(* general cam lock ctrl *)
FUNCTION_BLOCK FB_MC2_CamCtrl
VAR_INPUT
	bLockCam			: BOOL;			(* set TRUE to lock Slave axis to Master axis using cam table *)
	eStartMode			: MC_StartMode;	(* start mode for cam *)
	eCamTableID			: MC_CAM_ID;	(* NC cam table ID *)
	sCamTableRef		: MC_CAM_REF;	(* cam table reference structure *)
	fMasterOffset		: LREAL;		(* master offset on cam lock *)
	fSlaveOffset		: LREAL;		(* slave offset on cam lock *)
	fMasterScaling		: LREAL;		(* master scaling *)
	fSlaveScaling		: LREAL;		(* slave scaling *)
	sCamInOptions		: ST_CamInOptions;	(* cam coupling options *)
END_VAR
VAR_IN_OUT
	sMasterAxis			: AXIS_REF;		(* master axis *)
	sSlaveAxis			: AXIS_REF;		(* slave axis *)
END_VAR
VAR_OUTPUT
	bCamLocked			: BOOL;			(* TRUE = cam locked *)
	bCamError			: BOOL;			(* TRUE = cam lock error *)
	nCamErrorID			: UDINT;		(* cam lock error code *)
	bCamTableReadOK		: BOOL;			(* TRUE = cam table loaded from NC *)
	bCamActive			: BOOL;			(* TRUE = cam plate active but not yet in use *)
	bCamInSync			: BOOL;			(* TRUE = cam plate active and in use *)
	bCamUnlockPulse		: BOOL;			(* TRUE = cam has been unlocked, one-shout pulse output *)
	nCamPoints			: UDINT;		(* no of cam points in NC cam table *)
	sCamInfo			: MC_CamInfoData;	(* cam info *)
END_VAR
VAR
	fbPhaseDelay		: TON;
	fbReadCamTable		: MC_ReadMotionFunction;
	fbEnableCamLock		: RS;
	bEnableCamLock		: BOOL;
	fbLockCam			: MC_CamIn;
	fbUnlockCam			: MC_CamOut;
	bCamReady			: BOOL;
	fbCamInfo			: MC_CamInfo;
	bCamInfoDone		: BOOL;
	fbUnlockEvent		: F_TRIG;
	fbUnlockPulse		: TP;
END_VAR
(*
-------------------------------------------------------------------------------------------------
Date		Version	Author	Comments
-------------------------------------------------------------------------------------------------
30/01/2015	3.00.00	PB		Initial release

-------------------------------------------------------------------------------------------------
*)
VAR // added by the converter: edge detectors and wires of the graphical bodies
    _w1 : BOOL;
END_VAR

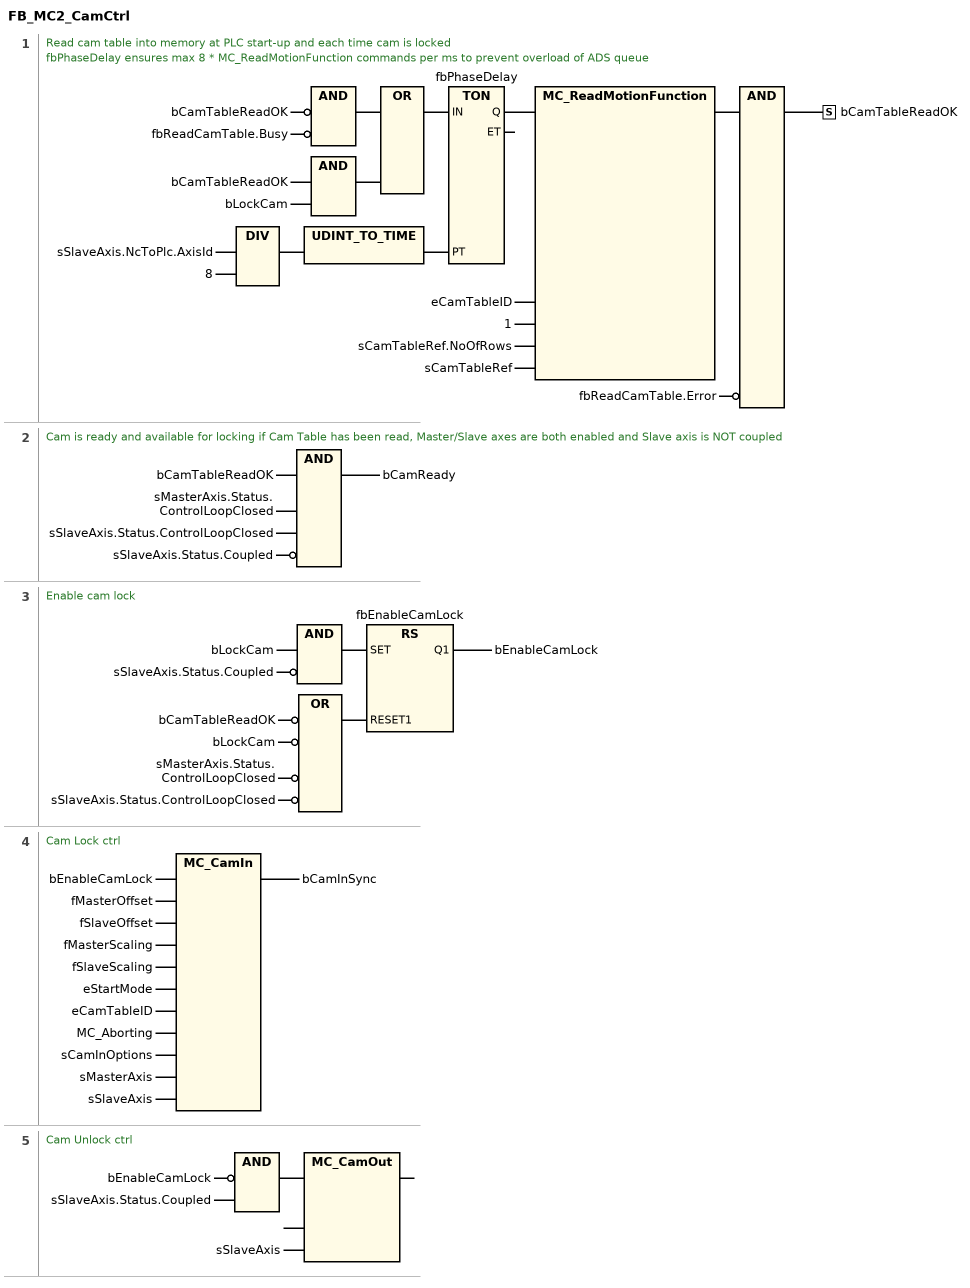
// NETWORK 1
// 					Read cam table into memory at PLC start-up and each time cam is locked
// fbPhaseDelay ensures max 8 * MC_ReadMotionFunction commands per ms to prevent overload of ADS queue
//
fbPhaseDelay(IN := NOT bCamTableReadOK AND NOT fbReadCamTable.Busy OR bCamTableReadOK AND bLockCam, PT := UDINT_TO_TIME(sSlaveAxis.NcToPlc.AxisId / 8)); // TON
bCamTableReadOK S= MC_ReadMotionFunction(fbPhaseDelay.Q, eCamTableID, 1, sCamTableRef.NoOfRows, sCamTableRef) AND NOT fbReadCamTable.Error;

// NETWORK 2
// Cam is ready and available for locking if Cam Table has been read, Master/Slave axes are both enabled and Slave axis is NOT coupled
bCamReady := bCamTableReadOK AND sMasterAxis.Status.ControlLoopClosed AND sSlaveAxis.Status.ControlLoopClosed AND NOT sSlaveAxis.Status.Coupled;

// NETWORK 3
// Enable cam lock
fbEnableCamLock(SET := bLockCam AND NOT sSlaveAxis.Status.Coupled, RESET1 := NOT bCamTableReadOK OR NOT bLockCam OR NOT sMasterAxis.Status.ControlLoopClosed OR NOT sSlaveAxis.Status.ControlLoopClosed); // RS
bEnableCamLock := fbEnableCamLock.Q1;

// NETWORK 4
// Cam Lock ctrl
bCamInSync := MC_CamIn(bEnableCamLock, fMasterOffset, fSlaveOffset, fMasterScaling, fSlaveScaling, eStartMode, eCamTableID, MC_Aborting, sCamInOptions, sMasterAxis, sSlaveAxis);

// NETWORK 5
// Cam Unlock ctrl
MC_CamOut(NOT bEnableCamLock AND sSlaveAxis.Status.Coupled, ???, sSlaveAxis);

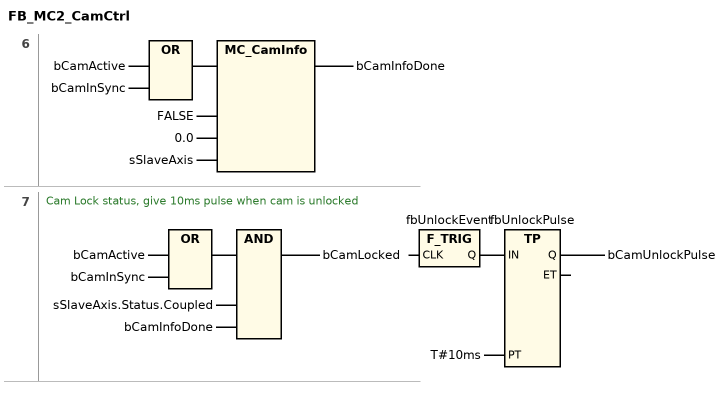
// NETWORK 6
bCamInfoDone := MC_CamInfo(bCamActive OR bCamInSync, FALSE, 0.0, sSlaveAxis);

// NETWORK 7
// Cam Lock status, give 10ms pulse when cam is unlocked
_w1 := (bCamActive OR bCamInSync) AND sSlaveAxis.Status.Coupled AND bCamInfoDone;
bCamLocked := _w1;
fbUnlockEvent(CLK := _w1); // F_TRIG
fbUnlockPulse(IN := fbUnlockEvent.Q, PT := T#10ms); // TP
bCamUnlockPulse := fbUnlockPulse.Q;

END_FUNCTION_BLOCK

(* stored: Version 1.1.0.1, ProductVersion 3.1.4024.15
   POU FB_MC2_CamCtrl: Id {2a460b83-a767-469a-a7b2-12d19a9edfed}, SpecialFunc None *)
